// Mitsubishi GX Works2 project: 201101二工位投板機20210324   PLC: FX3U/FX3UC
// HMI

// global labels: D
VAR_GLOBAL
  DSt1Dly AT D200 : INT;  (* Need to set *)
  DXferPosA AT D202 : DINT;  (* Need to set *)
  DXferPosB AT D204 : DINT;  (* Need to set *)
  DXferSpd AT D206 : DINT;  (* Need to set *)
  DXferPos AT D208 : DINT;  (* Need to set *)
  DVcDly AT D210 : INT;  (* Need to set *)
  DShockCnt AT D212 : INT;  (* Need to set *)
  DPls1Acc AT D8348 : INT;
  DPls1Dec AT D8349 : INT;
  DNowPos AT D8340 : DINT;
  DPls1Acc1 AT D214 : INT;  (* Need to set *)
  DPls1Dec1 AT D216 : INT;  (* Need to set *)
  DShock AT D218 : INT;
  DOverPos AT D220 : DINT;  (* Need to set *)
  DErrCode AT D7000 : INT;
  DWarningCode AT D7002 : INT;
  DSizeAPort AT D7004 : INT;
  DSizeBPort AT D7006 : INT;
  DStatus AT D7008 : INT;
  DSetPCBcountAPort AT D100 : INT;
  DNowCountAPort AT D102 : INT;
  DSetPCBcountBPort AT D104 : INT;
  DNowCountBPort AT D106 : INT;
  DShockTime AT D222 : INT;
  DXferDrop AT D224 : INT;
END_VAR

// global labels: IN
VAR_GLOBAL
  EMS1 AT X000 : BOOL;  (* 緊急停止鈕 *)
  STOP1 AT X001 : BOOL;  (* 停止鈕 *)
  Start1 AT X002 : BOOL;  (* 啟動紐 *)
  XFER_HOME_POS AT X011 : BOOL;  (* 移載原點 *)
  XFER_REV_POS AT X012 : BOOL;  (* 移載後極限 *)
  XFER_UP1_POS AT X013 : BOOL;  (* 移載氣缸上限 *)
  XFER_DN1_POS AT X014 : BOOL;  (* 移載氣缸下限 *)
  XFER_DN_OV AT X015 : BOOL;  (* 移載過壓 *)
  XFER_VC AT X016 : BOOL;  (* 吸版真空到達 *)
  AIR AT X017 : BOOL;  (* 氣壓壓力 *)
  XFER_FWD_POS AT X010 : BOOL;  (* 移載前極限 *)
  ST1_FEED_POS AT X021 : BOOL;  (* 置料有料上定位光電(NC)1 *)
  ST1_UP_POS AT X022 : BOOL;  (* 置料無料上極限開關1 *)
  ST1_POS AT X024 : BOOL;  (* 置料下限1 *)
  ST1_DN_POS AT X025 : BOOL;  (* 置料下極限1 *)
  ST1_AL AT X026 : BOOL;  (* 置料昇降馬達異常1 *)
  ST1_TABLE AT X027 : BOOL;  (* 棧板檢知光電1 *)
  ST2_FEED_POS AT X031 : BOOL;  (* 置料有料上定位光電(NC)2 *)
  ST2_UP_POS AT X032 : BOOL;  (* 置料無料上極限開關2 *)
  ST2_POS AT X034 : BOOL;  (* 置料下限2 *)
  ST2_DN_POS AT X035 : BOOL;  (* 置料下極限2 *)
  ST2_AL AT X036 : BOOL;  (* 置料昇降馬達異常2 *)
  ST2_TABLE AT X037 : BOOL;  (* 棧板檢知光電2 *)
  APR_AL AT X040 : BOOL;  (* 欠相保護器異常輸入 *)
  SDR1_AL AT X041 : BOOL;  (* 移載伺服異常 *)
  SDR1_RES AT X042 : BOOL;  (* 移載伺服重置 *)
  XFER_UP2_POS AT X044 : BOOL;  (* 移載氣缸2上限 *)
  XFER_DN2_POS AT X045 : BOOL;  (* 移載氣缸2下限 *)
  ST1_UP_PB AT X046 : BOOL;  (* 置料上升按鈕1 *)
  ST1_DN_PB AT X047 : BOOL;  (* 置料下降按鈕1 *)
  ST2_UP_PB AT X050 : BOOL;  (* 置料上升按鈕2 *)
  ST2_DN_PB AT X051 : BOOL;  (* 置料下降按鈕2 *)
  LINK1 AT X056 : BOOL;  (* 外部連線信號2 *)
  LINK2 AT X057 : BOOL;  (* 外部連線信號1 *)
  DoorAl AT X052 : BOOL;  (* 門檢 *)
END_VAR

// global labels: M
VAR_GLOBAL
  AT_ON AT M100 : BOOL;
  Alarm_No1 AT K8M200 : DINT;
  MEmgStop AT M98 : BOOL;
  MEmgReset AT M99 : BOOL;
  MGoHome AT M10 : BOOL;
  MHomeFinish AT M1990 : BOOL;
  MSizeReg AT M0 : BOOL;
  MGoPos AT M1 : BOOL;
  MPosFinish AT M1950 : BOOL;
  MOneRun AT M3 : BOOL;
  MAutoRun AT M4 : BOOL;
  MStopRun AT M97 : BOOL;
  MStopOk AT M100 : BOOL;
  MJog_Start AT M500 : BOOL;
  MJog_Stop AT M999 : BOOL;
  MJogTransferHome AT M400 : BOOL;
  MJogTransferPos1 AT M401 : BOOL;
  MJogTransferPos2 AT M402 : BOOL;
  MJogTransferB AT M13 : BOOL;
  MJogTransferF AT M12 : BOOL;
  MJogInCylinder AT M12 : BOOL;
  MJogOutCylinder AT M406 : BOOL;
  MJogVacOn AT M17 : BOOL;
  MJogVacBk AT M26 : BOOL;
  MXferFin AT M8029 : BOOL;
  LPosA AT M260 : BOOL;
  LPosB AT M261 : BOOL;
  MShock AT M250 : BOOL;
  MXferFinY0 AT M8340 : BOOL;
  LPosALack AT M267 : BOOL;
  LPosBLack AT M268 : BOOL;
  LOverPos AT M264 : BOOL;
  LRun AT M263 : BOOL;
  LChange AT M266 : BOOL;
  MJogOutShake1 AT M24 : BOOL;
  MJogOutShake2 AT M23 : BOOL;
  MJogLoader1Up AT M411 : BOOL;
  MJogLoader1Dn AT M412 : BOOL;
  MJogLoader2Up AT M413 : BOOL;
  MJogLoader2Dn AT M414 : BOOL;
  LEMS AT M269 : BOOL;
  MACntFin AT M12 : BOOL;
  MBCntFin AT M13 : BOOL;
  LAOnce AT M270 : BOOL;
  LBOnce AT M271 : BOOL;
  LStop AT M273 : BOOL;
END_VAR

// global labels: OUT
VAR_GLOBAL
  Pls1 AT Y000 : BOOL;  (* 移載CW *)
  Dir1 AT Y002 : BOOL;  (* 移載CCW *)
  SON AT Y004 : BOOL;  (* 移載SON *)
  RES AT Y005 : BOOL;  (* 移載RES *)
  O_XFER_UP1 AT Y011 : BOOL;  (* 吸盤氣缸1上升 *)
  O_XFER_DN1 AT Y012 : BOOL;  (* 吸盤氣缸1下降 *)
  O_XFER_VC_ON AT Y013 : BOOL;  (* 吸盤真空ON *)
  O_XFER_VC_OFF AT Y014 : BOOL;  (* 吸盤真空OFF *)
  O_XFER_VC_BK AT Y015 : BOOL;  (* 吸盤破真空 *)
  O_ST1_UP AT Y016 : BOOL;  (* 置料上升1 *)
  O_ST2_UP AT Y020 : BOOL;  (* 置料上升2 *)
  O_ST2_DN AT Y021 : BOOL;  (* 置料下降2 *)
  O_XFER_UP2 AT Y022 : BOOL;  (* 吸盤氣缸2上升 *)
  O_XFER_DN2 AT Y023 : BOOL;  (* 吸盤氣缸2下降 *)
  O_XFER_BLOW AT Y024 : BOOL;  (* 吹氣 *)
  O_XFER_SHOCK1 AT Y025 : BOOL;  (* 振動氣缸1 *)
  O_XFER_SHOCK2 AT Y026 : BOOL;  (* 振動氣缸2 *)
  O_START_LAMP AT Y027 : BOOL;  (* 啟動燈 *)
  O_STOP_LAMP AT Y030 : BOOL;  (* 停止燈 *)
  O_ST1_LAMP AT Y031 : BOOL;  (* 置料上升燈1 *)
  O_ST2_LAMP AT Y032 : BOOL;  (* 置料上升燈2 *)
  O_BZ AT Y033 : BOOL;  (* 塔燈-蜂鳴器 *)
  O_RL AT Y034 : BOOL;  (* 塔燈-紅燈 *)
  O_YL AT Y035 : BOOL;  (* 塔燈-黃燈 *)
  O_GL AT Y036 : BOOL;  (* 塔燈-綠燈 *)
  O_LINK1 AT Y037 : BOOL;  (* 放板完成 *)
  O_ST1_DN AT Y017 : BOOL;  (* 置料下降1 *)
END_VAR

// global labels: TandC
VAR_GLOBAL
  T_start AT TC0 : BOOL;
  TStartRun AT TS0 : BOOL;
  TStDlyRun AT TS1 : BOOL;
  TStDly AT TC1 : BOOL;
  TVcDly AT TC2 : BOOL;
  TVcDlyRun AT TS2 : BOOL;
  CShock AT CC1 : BOOL;
  CShockRun AT CS1 : BOOL;
END_VAR

// task Task_01 (event TRUE, interval 0, priority 31): POU_01

PROGRAM POU_01
	 DPls1Acc:=DPls1Acc1;
DPls1Dec:=DPls1Dec1;
LOverPos:=DNowPos>DOverPos;


set(MEmgStop,M300);
rst(MEmgReset,M300);
SET(M8043,M450);
RST(EMS1,M450);

M0 := OUT_T(NOT EMS1,T_START,30);
SON:= NOT (Alarm_No1>0) AND NOT EMS1 ;
RES:=NOT AT_ON AND (Alarm_No1>0) ;
rst(EMS1,AT_ON);
RST(Alarm_No1>0,AT_ON);
RST(Alarm_No1>0,LRun);
rst(ldp(TRUE,LEMS),LRun);
M8349:=EMS1;

O_RL:=M8013 AND Alarm_No1 >0 ;
O_BZ:=M8013 AND Alarm_No1 >0 ;
O_GL:= AT_ON OR (Alarm_No1=0 AND D50=2 AND  M8013) ;
O_YL:= D50=3;
MOVP(AT_ON,2,D40);
OUT(((Alarm_No1>0) AND NOT AT_ON AND M8013 ) OR AT_ON ,O_START_LAMP);

IF AT_ON AND Alarm_No1 = 0 THEN D110:=3 ; END_IF;
IF Alarm_No1 > 0 THEN D110:=4 ; END_IF;
IF NOT AT_ON AND Alarm_No1 = 0 THEN D110:=0 ; END_IF;
IF ST1_TABLE THEN D112:=100;ELSE D112:=0;END_IF;
IF ST2_TABLE THEN D114:=10;ELSE D114:=0;END_IF;		
D7008:= D110 + D112 + D114;

	
	
	
	

(*	 手動輸出	*)
IF TStartRun THEN 
	IF  NOT at_on (*AND (alarm_NO1 =0)*) THEN  	
	 	OUT((MJogLoader1Up OR ( ST1_UP_PB AND NOT ST1_DN_PB )) AND NOT ST1_UP_POS AND ST1_FEED_POS,O_ST1_UP);
	 	OUT((MJogLoader1Dn OR  (ST1_DN_PB AND NOT ST1_UP_PB )) AND NOT ST1_DN_POS,O_ST1_DN);
	 	OUT((MJogLoader2Up OR (ST2_UP_PB AND NOT ST2_DN_PB) ) AND NOT ST2_UP_POS AND ST2_FEED_POS,O_ST2_UP);
	 	OUT((MJogLoader2Dn OR( ST2_DN_PB AND NOT ST2_UP_PB)) AND NOT ST2_DN_POS,O_ST2_DN);
	 	DZRN( MJogTransferHome AND   XFER_UP1_POS AND   XFER_REV_POS,6000,200,XFER_HOME_POS,Pls1);
	 	DDRVA(MJogTransferPos1  AND   XFER_UP1_POS AND   XFER_REV_POS ,DXferPosA,DXferSpd,Pls1,Dir1);
		DDRVA(MJogTransferPos2  AND   XFER_UP1_POS AND   XFER_FWD_POS ,DXferPosB ,DXferSpd,Pls1,Dir1);
		DDRVI((MJogTransferB OR (ST2_UP_PB AND ST2_DN_PB))  AND  XFER_UP1_POS  AND XFER_REV_POS,-99999999,5000,Pls1,Dir1);
		DDRVI(( MJogTransferF OR (ST1_UP_PB AND ST1_DN_PB))  AND   XFER_UP1_POS  AND  XFER_FWD_POS  ,99999999,5000,Pls1,Dir1);			

		OUT(MJogInCylinder,O_XFER_DN1);
		OUT(MJogInCylinder,O_XFER_DN2);
		OUT(MJogVacOn,O_XFER_VC_ON);
		OUT(MJogVacBk,O_XFER_VC_BK);
		OUT(MJogOutShake1,O_XFER_SHOCK1);
		OUT(MJogOutShake2,O_XFER_SHOCK2);		
		RST (LDF(TRUE,MXferFinY0),MJogTransferHome );
		RST (LDF(TRUE,MXferFinY0),MJogTransferPos1 );
		RST (LDF(TRUE,MXferFinY0),MJogTransferPos2 );				



	END_IF;


(*ALTP(Start1,AT_ON);*)
OUT_T(Start1,TC12,3);
RST(TS12,AT_ON);
SET(LDP(TRUE,LRun)  OR (LDP(TRUE,Start1) )  AND Alarm_No1=0 ,AT_ON);

RST(LDP(TRUE,LEMS)OR (LDP(TRUE,Start1) ) AND Alarm_No1>0,AT_ON);


RST(  D3=121 AND lstop , AT_ON );
RST ( D3=121 AND lstop , LStop );
RST(D3=131  , AT_ON );
RST(D3=131  , LStop );

RST ( LDF(TRUE,AT_ON), M1);
RST ( LDF(TRUE,AT_ON), M2);

RST(D3=131 AND lstop AND  (( NOT M1 AND NOT M2 ) OR ((D1=2 AND LDF(TRUE,M1) ) OR( D2=2 AND LDF(TRUE,M2) ))) , AT_ON );
RST(D3=131 AND lstop AND  (( NOT M1 AND NOT M2 ) OR ((D1=2 AND LDF(TRUE,M1) ) OR( D2=2 AND LDF(TRUE,M2) )))  , LStop );

RST(LDP(TRUE,Start1),D240);

RST(LDP(TRUE,AT_ON),LStop);
RST((LDP(TRUE,LEMS)) OR (LDF(TRUE,AT_ON)) ,LPosA);
RST((LDP(TRUE,LEMS)) OR (LDF(TRUE,AT_ON)) ,LPosB);
RST((LDP(TRUE,LEMS)) OR (LDF(TRUE,AT_ON)) ,LStop);
ZRSTP(AT_ON,D100,D107);

IF LDP(TRUE,AT_ON) THEN D1:=3; D2:=3; D3:=1;DShock:=0;D240:=0;END_IF;
IF LDF(TRUE,AT_ON) THEN D1:=0; D2:=0; D3:=0; 
	RST(TRUE,MXferFinY0);
	 zrst(TRUE ,Y11,Y26);
	 T20 :=0;	
	 RST(TS20,T20);
	 RST(TRUE,LRun);
	 END_IF;

OUT_T(LEMS,TC8,5);
RST(TS8,LEMS);

	
ZRSTP(NOT ems1,Y11,Y26);


(*out((AT_ON OR (NOT AT_ON AND M8013)) ,O_GL);
out((( Alarm_No1 > 0 )  AND M8013)  ,O_RL);
out(((  Alarm_No1 > 0)  AND M8013) ,O_BZ);*)

DINCP((M10 OR M11) AND D3=6,D250);
DINCP(M10 AND D3=6,D252);
DINCP(M11 AND D3=6,D254);


(*	 A疊料自動 *)

IF at_on THEN 
	 	CASE  D1 OF
		1:
		OUT (NOT ST1_DN_POS AND  D1=1  ,O_ST1_DN);
		 IF  ST1_DN_POS THEN D1:=2;  END_IF;
		2 :
		RST(TRUE,M1);
		OUT (NOT ST1_UP_PB AND M8013,O_ST1_LAMP); 
	 	IF ST1_UP_PB THEN D1 := 3; SET(TRUE ,LPosA) ; END_IF;

	 	    
	 	3 :
           OUT_T(D1=3 AND ST1_FEED_POS AND NOT ST1_UP_POS AND LPosA ,TC10,D204);
	 		OUT (D1=3 AND TS10 AND ST1_TABLE ,O_ST1_UP); 	 
	 	(*IF NOT ST1_FEED_POS AND D3=10 THEN D1:= 5;  END_IF ;*)
	 		IF (ST1_UP_POS OR NOT ST1_TABLE) AND LPosA  THEN D1:=10; END_IF; 
	 	4 :
	 	OUT ( NOT ST1_FEED_POS OR NOT ST1_UP_POS ,O_ST1_UP); 
	 	IF  ST1_FEED_POS THEN D1:= 5;  END_IF ;
	 	IF ST1_UP_POS THEN D1:=1;END_IF;
	 	5:
	 	IF D3=10 AND LPosA AND XFER_UP1_POS AND XFER_UP2_POS THEN D1:= 3;  ; END_IF ;
	 	6 : 
	 	OUT_T(NOT TStDlyRun,TStDly,DSt1Dly);
	 	OUT (NOT TStDlyRun,O_ST1_DN);
	 	IF TStDlyRun THEN D1:= 3; rst(TStDlyRun,TStDly);RST(TStDlyRun,T1);  END_IF ;
		10:
		RST (TRUE,O_ST1_UP); 
		OUT (NOT ST1_DN_POS,O_ST1_DN); 
		SET(TRUE,M1);
		
		 IF  ST1_DN_POS THEN D1:=2;   END_IF;	 		
	END_CASE;
	 	END_IF;
	 	

(*RST(LDP(TRUE,D1=10),LPosA);	 	*)
 	
	 	
(*	 B疊料自動 *)  

IF at_on THEN 
	 	CASE  D2 OF
		1:
		    OUT (NOT ST2_DN_POS AND  D2=1,O_ST2_DN); 	
		 IF ST2_DN_POS THEN D2:=2; END_IF;
		2 :
		RST(TRUE,M2);
		OUT (NOT ST2_UP_PB AND M8013,O_ST2_LAMP);
	 	IF ST2_UP_PB THEN D2 := 3; SET(TRUE ,LPosB) ;  END_IF;
	 	3 :
	 	        OUT_T(D2=3 AND ST2_FEED_POS AND NOT ST2_UP_POS AND LPosB,TC11,D204);
	 		OUT (D2=3 AND TS11 AND ST2_TABLE,O_ST2_UP); 	
	 	(*IF NOT ST2_FEED_POS AND D3=10 THEN D2:= 5;  END_IF ;*)
	 	IF (ST2_UP_POS OR NOT ST2_TABLE) AND LPosB  THEN D2:=10; END_IF; 
	 	4 :
	 	OUT (  NOT ST2_FEED_POS OR NOT ST2_UP_POS ,O_ST2_UP);
	 	IF ST2_FEED_POS THEN D2:= 5;  END_IF ;	 
	 	IF ST2_UP_POS THEN D2:=1;END_IF;
	 	5 :
	 	IF D3=10 AND LPosB  AND XFER_UP1_POS AND XFER_UP2_POS  THEN D2:= 3;  ; END_IF ;
	 	6 : 
	 	OUT_T(NOT TStDlyRun,TStDly,DSt1Dly );
	 	 OUT (NOT TStDlyRun,O_ST2_DN);
	 	IF TStDlyRun THEN D2:= 3; rst(TStDlyRun,TStDly);RST(TStDlyRun,T1);    END_IF ;
		10:
		RST (TRUE,O_ST2_UP); 
		SET(TRUE,M2);
		OUT (NOT ST2_DN_POS,O_ST2_DN); 
		
		 IF  ST2_DN_POS THEN D2:=2;  END_IF;	 		
	END_CASE;
	 	END_IF;
    

(*RST(LDP(TRUE,D2=10),LPosB); 	*)
	 		 	
PLS(D1=10,M300);	 	
PLS(D2=10,M301);

(*	 AB疊料自動順序 *)

M10:=LPosA AND NOT M11;
M11:=LPosB AND NOT M10;
 	
(*放版動作*)
IF at_on THEN 
	 	CASE  D3 OF
		1:
		 out(NOT  XFER_UP1_POS ,O_XFER_UP1);
		 out( NOT  XFER_UP2_POS,O_XFER_UP2);
		 IF XFER_UP1_POS AND XFER_UP2_POS THEN   D3:=2;END_IF;
		2 :
	 	 IF LDF(TRUE,MXferFinY0) THEN D3 := 3; END_IF;
	 	3 :
	 	RST(NOT XFER_UP2_POS,O_XFER_DN2);
	 	IF M10 AND D1 =3 AND NOT LStop THEN D3:= 4; END_IF ;
	 	IF M11 AND D2 =3 AND NOT LStop THEN D3:= 100; END_IF ;
	 	IF M10  AND D1=10  AND DNowPos = DXferPos THEN D3:=101; END_IF;
	 	IF M11  AND D2=10  AND DNowPos = DXferPos THEN D3:=101; END_IF;	 		
	 	IF NOT LPosA  AND NOT LPosB THEN D3:=120; END_IF;
	 	IF LStop THEN D3:=130; END_IF;	 		
	 	4 :
	 	IF  LDF(TRUE,MXferFinY0) THEN D3:= 110; END_IF ;
	 	100 :
	 	IF  LDF(TRUE,MXferFinY0) THEN D3:= 110; END_IF ;
	 	101:
	 	IF  LDF(TRUE,MXferFinY0)  THEN D3:= 103; END_IF ;
	 	103:
	 	IF  LPosA OR LPosB THEN D3:= 3; END_IF ;	 		 		
	 	102:
	 	IF  LDP(TRUE,ST1_DN_POS) OR LDp(TRUE,ST2_DN_POS)  THEN D3:= 3; END_IF ;	 		
	 	110:
	 	IF (M10 AND NOT ST1_FEED_POS )  OR	(M11 AND NOT ST2_FEED_POS) THEN D3:=5 ;END_IF;
	 	120:
	 	IF  LDF(TRUE,MXferFinY0)  THEN D3:= 121; END_IF ; 		 	
	 	121:
	 	IF  LDP(TRUE,LPosA) OR LDP(TRUE,LPosB)  THEN D3:= 3; END_IF ;
	 	130:
	 	IF  LDF(TRUE,MXferFinY0)  THEN D3:= 131; END_IF ; 		 	
	 	131:
	 	IF  LDP(TRUE,LPosA) OR LDP(TRUE,LPosB)  THEN D3:= 3; END_IF ;	 		
	 		
	 		 
 				 	 		
	 	5 : 
	 	 out(TRUE,O_XFER_DN1);
		
	 	IF XFER_DN1_POS THEN D3:= 6;   END_IF ;
	 	6 : 
	 	 out(TRUE,O_XFER_DN1);
	 	OUT (TRUE,O_XFER_VC_ON); 

	 	
	 	IF XFER_VC THEN D3:= 7; END_IF ;
	 	7 : 
	 	OUT_T(D3=7,TVcDly,DVcDly);
	 	IF TVcDlyRun THEN D3:= 200 ;rst(TVcDlyRun,TVcDly);rst(TVcDlyRun,T2);END_IF ;
	 	200:	
	 	RST(NOT XFER_UP1_POS,O_XFER_DN1);
		RST(NOT XFER_UP2_POS,O_XFER_DN2);
	 	IF XFER_UP1_POS AND XFER_UP2_POS  THEN   D3:=8;END_IF;
	 			
	 		
	 		
	 		
	 	8 : 
	 	out(MShock  ,O_XFER_SHOCK1);
	 	out(NOT MShock,O_XFER_SHOCK2);
	 	INCP(MShock,DShock);
	 	IF D218 > DShockCnt THEN D3:= 201;CN1:=0;DShock:=0;rst(TRUE,O_XFER_SHOCK1);rst(TRUE,O_XFER_SHOCK2);
	 	END_IF ;
	
	 	201:
	 	SET(TRUE,O_XFER_DN1);
		IF XFER_DN1_POS   THEN   D3:=202;END_IF;	
		202:	
		RST(TRUE,O_XFER_DN1);
		IF XFER_UP1_POS   THEN   D3:=203;END_IF;	
	 	203:
	 	SET(TRUE,O_XFER_DN1);
		IF XFER_DN1_POS   THEN   D3:=9;END_IF;				


	 	9 : 
		RST(NOT XFER_UP1_POS,O_XFER_DN1); 	
		IF NOT XFER_VC THEN D3:=5;END_IF;
		IF XFER_UP1_POS   AND LINK1 AND LINK2 THEN   D3:=10;  out( TRUE,O_XFER_DN2);D240:=0;END_IF;
		(*link1=X56=run  LINK2=X57=LOCK CYNDER UPPER  *)
	 	10 : 
	 	out( TRUE,O_XFER_DN2);
	 	IF  LDF(TRUE,MXferFinY0)THEN   D3:= 11;   END_IF ;
	 	11 : 
	 	out(TRUE,O_XFER_DN1);
		 out( TRUE,O_XFER_DN2);
	 	IF XFER_DN1_POS AND XFER_DN2_POS THEN D3:= 12;   END_IF ;
	 	12  : 
	 	OUT_T(NOT TS6,TC6,DXferDrop);
	 	(*out(NOT TS6,O_XFER_VC_OFF);*)
	 	rst(TRUE,O_XFER_VC_ON);
	 	IF TS6 THEN D3:= 13 ;rst(TS6,TC6); rst(TS6,T6); END_IF ;
	 	13  : 
	 	OUT_T(NOT TS7,TC7,DXferDrop);
	 	 OUT(TRUE,O_XFER_VC_BK);
	 	IF TS7 THEN D3:= 14 ;rst(TS7,TC7);rst(TS7,T7);  END_IF ;
	 	14  :  	

		RST(NOT XFER_UP1_POS,O_XFER_DN1);
		RST(NOT XFER_UP2_POS,O_XFER_DN2);
		 RST(NOT XFER_UP1_POS AND NOT XFER_UP2_POS,O_XFER_VC_BK);
	 	IF XFER_UP1_POS  THEN D3:= 3; END_IF ;
	   (* IF XFER_UP1_POS AND  XFER_UP2_POS THEN D3:= 3; END_IF ;*)	 		
	 	15  : 
	 	IF XFER_VC THEN D3:= 16;  ELSE O_BZ :=TRUE;END_IF ;
	 	16  : 
	 	IF XFER_VC THEN D3:= 17;  ELSE O_BZ :=TRUE;END_IF ;
	 	17  : 
	 	IF XFER_VC THEN D3:= 18;  ELSE O_BZ :=TRUE;END_IF ;
	 	18  : 
	 	IF XFER_VC THEN D3:= 19;  ELSE O_BZ :=TRUE;END_IF ;

	 	END_CASE;
	 	
LPosALack	:= NOT  D1=3; 	
LPosBLack := NOT  D2=3;


MACntFin := DNowCountAPort <= DSetPCBcountAPort   ;
MBCntFin := DNowCountBPort <= DSetPCBcountBPort   ;
INCP( D3=12,DNowCountAPort);
(* INCP(M11 AND D3=13,DNowCountBPort);	 *)	
RST(D3=1,DNowCountAPort);
RST(D3=1,DNowCountBPort);
RST(LAOnce AND D3=13  ,LAOnce);
RST(LBOnce AND D3=13  ,LBOnce);

END_IF;
OUT(AT_ON AND NOT LOverPos AND NOT  Dir1 AND Pls1 AND ( D3=4 OR D3=100 OR D3=10 OR D3=101 OR D3=120 OR D3=130 ) ,  O_LINK1 );

	 	END_IF;(*開機延遲啟動*)
	 	(*歸零方向指定*)
	 	M8342:=M600;
	
	 	 DZRN(D3= 2,6000,200,XFER_HOME_POS,Pls1);
	 	DDRVA(D3= 4,DXferPosA,DXferSpd,Pls1,Dir1); 
	 	DDRVA(D3= 100,DXferPosB,DXferSpd,Pls1,Dir1) ; 	
	 	DDRVA(D3= 10,DXferPos,DXferSpd,Pls1,Dir1) ;
	 	DDRVA(D3= 101,200,DXferSpd,Pls1,Dir1) ;
	 	DDRVA(D3= 120,210,DXferSpd,Pls1,Dir1) ;
	 	DDRVA(D3= 130,205,DXferSpd,Pls1,Dir1) ;


(*0.5秒震動*)
IF D3=8 THEN 
out_t(TRUE,TC4,D222);
out_t(TS4,TC5,D222);
out(TS4,MShock);
RST(TS5,TC4);
END_IF;

(*真空超時*)
M16:=D3=6;
OUT_T ( M16 ,TC25,30);
IF TS25 THEN D7000:=9;END_IF;
SET(TS25,M219);
RST(TS25,TC25);

(*吸版次數過多*)
IF D240 >3 THEN M226:=TRUE;D7000:=12;END_IF;
INCP(D3=9,D240);

(*氣壓源無氣壓*)
IF AIR  THEN 
	M216 := TRUE;D7000:=8;
END_IF; 

 (*無棧板*)
 IF ((NOT st1_table AND LPosA)  OR ( NOT ST2_TABLE AND LPosB) )  AND  LDP(TRUE,at_on) THEN
	M214 := TRUE;D7000:=7;
 END_IF;
 
  (*移動中掉版*)
IF AT_ON AND D3=10  AND NOT XFER_VC THEN
	M225 := TRUE;D7000:=10;
END_IF;
  (*移動超時*)
IF Pls1 AND AT_ON THEN
	OUT_T (TRUE,TC20,K150);
IF TS20 = TRUE THEN 	M208:=TRUE;D7000:=6; 
	END_IF;
ELSE
	T20 :=0;
	RST(TS20,T20); 
END_IF;



zrst(  ( Alarm_No1>0 AND (LDP(TRUE,LEMS) OR ldp(TRUE,Start1))   ) OR  LDF(TRUE,EMS1) ,M200,M232);
rst(LDP(TRUE,LEMS)  OR LDP(TRUE,Start1),D7000);

IF EMS1 OR MEmgStop  THEN M200:=TRUE;D7000:=1;
END_IF;
IF TStartRun THEN
(*
IF NOT XFER_DN_OV =TRUE THEN M201:=TRUE;
END_IF;
*)
IF ST1_AL = TRUE THEN M202:=TRUE;D7000:=2;
END_IF;

IF ST2_AL = TRUE THEN M203:=TRUE;D7000:=3;
END_IF;

IF APR_AL = TRUE THEN M204:=TRUE;D7000:=4;
END_IF;

IF NOT SDR1_AL =TRUE THEN M205:=TRUE;D7000:=5;
END_IF;
	
IF NOT DoorAl THEN M206:=TRUE ; D7000:=11;END_IF;	

END_IF;
END_PROGRAM
